// Geometric and Coordinate Transformations
NodeFactory.AddNodeAsPrototype('Vision/Geometric and Coordinate Transformations/Calibration/F_VN_CalibrateCamera', node_F_VN_CalibrateCamera);
//NodeFactory.AddNodeAsPrototype('Vision/Geometric and Coordinate Transformations/Calibration/F_VN_CalibrateCameraExp', node_F_VN_CalibrateCameraExp);
//NodeFactory.AddNodeAsPrototype('Vision/Geometric and Coordinate Transformations/Calibration/F_VN_CalibrateCameraExp2', node_F_VN_CalibrateCameraExp2);
//NodeFactory.AddNodeAsPrototype('Vision/Geometric and Coordinate Transformations/Calibration/F_VN_CalibrateCameraExp3', node_F_VN_CalibrateCameraExp3);
NodeFactory.AddNodeAsPrototype('Vision/Geometric and Coordinate Transformations/Calibration/F_VN_CalibrateCameraManually', node_F_VN_CalibrateCameraManually);
NodeFactory.AddNodeAsPrototype('Vision/Geometric and Coordinate Transformations/Calibration/F_VN_CalibrateCameraManuallyExp', node_F_VN_CalibrateCameraManuallyExp);
NodeFactory.AddNodeAsPrototype('Vision/Geometric and Coordinate Transformations/Calibration/F_VN_CalibrateCameraPlanar', node_F_VN_CalibrateCameraPlanar);
NodeFactory.AddNodeAsPrototype('Vision/Geometric and Coordinate Transformations/Calibration/F_VN_CalibrateCameraPlanarExp', node_F_VN_CalibrateCameraPlanarExp);
//NodeFactory.AddNodeAsPrototype('Vision/Geometric and Coordinate Transformations/Calibration/F_VN_CalibrateLinescanCamera', node_F_VN_CalibrateLinescanCamera);
//NodeFactory.AddNodeAsPrototype('Vision/Geometric and Coordinate Transformations/Calibration/F_VN_CalibrateLinescanCameraExp', node_F_VN_CalibrateLinescanCameraExp);
NodeFactory.AddNodeAsPrototype('Vision/Geometric and Coordinate Transformations/Calibration/F_VN_CompensateLensDistortion', node_F_VN_CompensateLensDistortion);
NodeFactory.AddNodeAsPrototype('Vision/Geometric and Coordinate Transformations/Calibration/F_VN_CompensateLensDistortionExp1', node_F_VN_CompensateLensDistortionExp1);
NodeFactory.AddNodeAsPrototype('Vision/Geometric and Coordinate Transformations/Calibration/F_VN_CompensateLensDistortionExp2', node_F_VN_CompensateLensDistortionExp2);
NodeFactory.AddNodeAsPrototype('Vision/Geometric and Coordinate Transformations/Calibration/F_VN_CompensateLensDistortionForPoints', node_F_VN_CompensateLensDistortionForPoints);
NodeFactory.AddNodeAsPrototype('Vision/Geometric and Coordinate Transformations/Calibration/F_VN_CompensateLensDistortionForPointsExp1', node_F_VN_CompensateLensDistortionForPointsExp1);
NodeFactory.AddNodeAsPrototype('Vision/Geometric and Coordinate Transformations/Calibration/F_VN_CompensateLensDistortionForPointsExp2', node_F_VN_CompensateLensDistortionForPointsExp2);
NodeFactory.AddNodeAsPrototype('Vision/Geometric and Coordinate Transformations/Calibration/F_VN_DetectPatternPoints', node_F_VN_DetectPatternPoints);
NodeFactory.AddNodeAsPrototype('Vision/Geometric and Coordinate Transformations/Calibration/F_VN_DetectPatternPointsExp', node_F_VN_DetectPatternPointsExp);
NodeFactory.AddNodeAsPrototype('Vision/Geometric and Coordinate Transformations/Calibration/F_VN_DetectPatternPoints2', node_F_VN_DetectPatternPoints2);
NodeFactory.AddNodeAsPrototype('Vision/Geometric and Coordinate Transformations/Calibration/F_VN_GenerateCalibrationPatternReferencePoints', node_F_VN_GenerateCalibrationPatternReferencePoints);
NodeFactory.AddNodeAsPrototype('Vision/Geometric and Coordinate Transformations/Calibration/F_VN_ImagePointsWorldDistance', node_F_VN_ImagePointsWorldDistance);
NodeFactory.AddNodeAsPrototype('Vision/Geometric and Coordinate Transformations/Calibration/F_VN_SolvePnP', node_F_VN_SolvePnP);
NodeFactory.AddNodeAsPrototype('Vision/Geometric and Coordinate Transformations/Calibration/F_VN_SolvePnPExp', node_F_VN_SolvePnPExp);
NodeFactory.AddNodeAsPrototype('Vision/Geometric and Coordinate Transformations/Calibration/F_VN_SortAxisAlignedPatternPoints', node_F_VN_SortAxisAlignedPatternPoints);
NodeFactory.AddNodeAsPrototype('Vision/Geometric and Coordinate Transformations/Calibration/F_VN_SortDetectedPatternPoints', node_F_VN_SortDetectedPatternPoints);
NodeFactory.AddNodeAsPrototype('Vision/Geometric and Coordinate Transformations/Calibration/F_VN_TransformCoordinatesImageToWorld_Container', node_F_VN_TransformCoordinatesImageToWorld_Container);
NodeFactory.AddNodeAsPrototype('Vision/Geometric and Coordinate Transformations/Calibration/F_VN_TransformCoordinatesImageToWorld_Point', node_F_VN_TransformCoordinatesImageToWorld_Point);
NodeFactory.AddNodeAsPrototype('Vision/Geometric and Coordinate Transformations/Calibration/F_VN_TransformCoordinatesPlanar_Container', node_F_VN_TransformCoordinatesPlanar_Container);
NodeFactory.AddNodeAsPrototype('Vision/Geometric and Coordinate Transformations/Calibration/F_VN_TransformCoordinatesPlanar_Point', node_F_VN_TransformCoordinatesPlanar_Point);
NodeFactory.AddNodeAsPrototype('Vision/Geometric and Coordinate Transformations/Calibration/F_VN_TransformCoordinatesWorldToImage_Container', node_F_VN_TransformCoordinatesWorldToImage_Container);
NodeFactory.AddNodeAsPrototype('Vision/Geometric and Coordinate Transformations/Calibration/F_VN_TransformCoordinatesWorldToImage_Point', node_F_VN_TransformCoordinatesWorldToImage_Point);
NodeFactory.AddNodeAsPrototype('Vision/Geometric and Coordinate Transformations/F_VN_AlignRotatedImageRegion', node_F_VN_AlignRotatedImageRegion);
NodeFactory.AddNodeAsPrototype('Vision/Geometric and Coordinate Transformations/F_VN_AlignRotatedImageRegionExp', node_F_VN_AlignRotatedImageRegionExp);
NodeFactory.AddNodeAsPrototype('Vision/Geometric and Coordinate Transformations/F_VN_ApplyRotationToAffineTransformation', node_F_VN_ApplyRotationToAffineTransformation);
NodeFactory.AddNodeAsPrototype('Vision/Geometric and Coordinate Transformations/F_VN_ApplyRotationToAffineTransformationExp', node_F_VN_ApplyRotationToAffineTransformationExp);
NodeFactory.AddNodeAsPrototype('Vision/Geometric and Coordinate Transformations/F_VN_ApplyScalingToAffineTransformation', node_F_VN_ApplyScalingToAffineTransformation);
NodeFactory.AddNodeAsPrototype('Vision/Geometric and Coordinate Transformations/F_VN_ApplyScalingToAffineTransformationExp', node_F_VN_ApplyScalingToAffineTransformationExp);
NodeFactory.AddNodeAsPrototype('Vision/Geometric and Coordinate Transformations/F_VN_ApplyTranslationToAffineTransformation', node_F_VN_ApplyTranslationToAffineTransformation);
NodeFactory.AddNodeAsPrototype('Vision/Geometric and Coordinate Transformations/F_VN_ApplyTranslationToAffineTransformationExp', node_F_VN_ApplyTranslationToAffineTransformationExp);
NodeFactory.AddNodeAsPrototype('Vision/Geometric and Coordinate Transformations/F_VN_ApplyYAxisInversionToAffineTransformation', node_F_VN_ApplyYAxisInversionToAffineTransformation);
NodeFactory.AddNodeAsPrototype('Vision/Geometric and Coordinate Transformations/F_VN_ApplyYAxisInversionToAffineTransformationExp', node_F_VN_ApplyYAxisInversionToAffineTransformationExp);
NodeFactory.AddNodeAsPrototype('Vision/Polarization/F_VN_DemosaicPolarizedImage', node_F_VN_DemosaicPolarizedImage);
NodeFactory.AddNodeAsPrototype('Vision/Polarization/F_VN_AngleAndDegreeOfLinearPolarization', node_F_VN_AngleAndDegreeOfLinearPolarization);
NodeFactory.AddNodeAsPrototype('Vision/Polarization/F_VN_PolarizedImageGlareReduction', node_F_VN_PolarizedImageGlareReduction);
NodeFactory.AddNodeAsPrototype('Vision/Geometric and Coordinate Transformations/F_VN_ConvertCartesianToPolarAngleImage', node_F_VN_ConvertCartesianToPolarAngleImage);
NodeFactory.AddNodeAsPrototype('Vision/Geometric and Coordinate Transformations/F_VN_ConvertCartesianToPolarAngleImageExp', node_F_VN_ConvertCartesianToPolarAngleImageExp);
NodeFactory.AddNodeAsPrototype('Vision/Geometric and Coordinate Transformations/F_VN_ConvertCartesianToPolarAngles', node_F_VN_ConvertCartesianToPolarAngles);
NodeFactory.AddNodeAsPrototype('Vision/Geometric and Coordinate Transformations/F_VN_ConvertCartesianToPolarAnglesExp', node_F_VN_ConvertCartesianToPolarAnglesExp);
NodeFactory.AddNodeAsPrototype('Vision/Geometric and Coordinate Transformations/F_VN_ConvertCartesianToPolarImages', node_F_VN_ConvertCartesianToPolarImages);
NodeFactory.AddNodeAsPrototype('Vision/Geometric and Coordinate Transformations/F_VN_ConvertCartesianToPolarImagesExp', node_F_VN_ConvertCartesianToPolarImagesExp);
NodeFactory.AddNodeAsPrototype('Vision/Geometric and Coordinate Transformations/F_VN_ConvertCartesianToPolarMagnitudeImage', node_F_VN_ConvertCartesianToPolarMagnitudeImage);
NodeFactory.AddNodeAsPrototype('Vision/Geometric and Coordinate Transformations/F_VN_ConvertCartesianToPolarMagnitudes', node_F_VN_ConvertCartesianToPolarMagnitudes);
NodeFactory.AddNodeAsPrototype('Vision/Geometric and Coordinate Transformations/F_VN_ConvertCartesianToPolarPoints', node_F_VN_ConvertCartesianToPolarPoints);
NodeFactory.AddNodeAsPrototype('Vision/Geometric and Coordinate Transformations/F_VN_ConvertCartesianToPolarPointsExp', node_F_VN_ConvertCartesianToPolarPointsExp);
NodeFactory.AddNodeAsPrototype('Vision/Geometric and Coordinate Transformations/F_VN_ConvertPolarToCartesianImages', node_F_VN_ConvertPolarToCartesianImages);
NodeFactory.AddNodeAsPrototype('Vision/Geometric and Coordinate Transformations/F_VN_ConvertPolarToCartesianImagesExp', node_F_VN_ConvertPolarToCartesianImagesExp);
NodeFactory.AddNodeAsPrototype('Vision/Geometric and Coordinate Transformations/F_VN_ConvertPolarToCartesianPoints', node_F_VN_ConvertPolarToCartesianPoints);
NodeFactory.AddNodeAsPrototype('Vision/Geometric and Coordinate Transformations/F_VN_ConvertPolarToCartesianPointsExp', node_F_VN_ConvertPolarToCartesianPointsExp);
NodeFactory.AddNodeAsPrototype('Vision/Geometric and Coordinate Transformations/F_VN_DecomposeAffineTransformation', node_F_VN_DecomposeAffineTransformation);
NodeFactory.AddNodeAsPrototype('Vision/Geometric and Coordinate Transformations/F_VN_DecomposeAffineTransformationExp', node_F_VN_DecomposeAffineTransformationExp);
NodeFactory.AddNodeAsPrototype('Vision/Geometric and Coordinate Transformations/F_VN_DecomposeHomography', node_F_VN_DecomposeHomography);
NodeFactory.AddNodeAsPrototype('Vision/Geometric and Coordinate Transformations/F_VN_DecomposeHomographyExp', node_F_VN_DecomposeHomographyExp);
NodeFactory.AddNodeAsPrototype('Vision/Geometric and Coordinate Transformations/F_VN_FlipImage', node_F_VN_FlipImage);
NodeFactory.AddNodeAsPrototype('Vision/Geometric and Coordinate Transformations/F_VN_GenerateAffineTransformationUnitMatrix2D', node_F_VN_GenerateAffineTransformationUnitMatrix2D);
NodeFactory.AddNodeAsPrototype('Vision/Geometric and Coordinate Transformations/F_VN_GetAffineTransformation', node_F_VN_GetAffineTransformation);
NodeFactory.AddNodeAsPrototype('Vision/Geometric and Coordinate Transformations/F_VN_GetAffineTransformation2D', node_F_VN_GetAffineTransformation2D);
//NodeFactory.AddNodeAsPrototype('Vision/Geometric and Coordinate Transformations/F_VN_GetAffineTransformation2DExp', node_F_VN_GetAffineTransformation2DExp);
NodeFactory.AddNodeAsPrototype('Vision/Geometric and Coordinate Transformations/F_VN_GetPerspectiveTransformation', node_F_VN_GetPerspectiveTransformation);
NodeFactory.AddNodeAsPrototype('Vision/Geometric and Coordinate Transformations/F_VN_Homography', node_F_VN_Homography);
NodeFactory.AddNodeAsPrototype('Vision/Geometric and Coordinate Transformations/F_VN_HomographyExp', node_F_VN_HomographyExp);
NodeFactory.AddNodeAsPrototype('Vision/Geometric and Coordinate Transformations/F_VN_InvertAffineTransformation', node_F_VN_InvertAffineTransformation);
NodeFactory.AddNodeAsPrototype('Vision/Geometric and Coordinate Transformations/F_VN_PerspectiveTransformation', node_F_VN_PerspectiveTransformation);
NodeFactory.AddNodeAsPrototype('Vision/Geometric and Coordinate Transformations/F_VN_PyramidDown', node_F_VN_PyramidDown);
NodeFactory.AddNodeAsPrototype('Vision/Geometric and Coordinate Transformations/F_VN_PyramidUp', node_F_VN_PyramidUp);
NodeFactory.AddNodeAsPrototype('Vision/Geometric and Coordinate Transformations/F_VN_ConvertMaps', node_F_VN_ConvertMaps);
NodeFactory.AddNodeAsPrototype('Vision/Geometric and Coordinate Transformations/F_VN_RemapImage', node_F_VN_RemapImage);
NodeFactory.AddNodeAsPrototype('Vision/Geometric and Coordinate Transformations/F_VN_RemapImageExp', node_F_VN_RemapImageExp);
NodeFactory.AddNodeAsPrototype('Vision/Geometric and Coordinate Transformations/F_VN_RemapImageToLogPolarSpace', node_F_VN_RemapImageToLogPolarSpace);
NodeFactory.AddNodeAsPrototype('Vision/Geometric and Coordinate Transformations/F_VN_RemapImageToLogPolarSpaceExp', node_F_VN_RemapImageToLogPolarSpaceExp);
NodeFactory.AddNodeAsPrototype('Vision/Geometric and Coordinate Transformations/F_VN_RemapImageToLogPolarSpaceExp2', node_F_VN_RemapImageToLogPolarSpaceExp2);
NodeFactory.AddNodeAsPrototype('Vision/Geometric and Coordinate Transformations/F_VN_RemapImageToPolarSpace', node_F_VN_RemapImageToPolarSpace);
NodeFactory.AddNodeAsPrototype('Vision/Geometric and Coordinate Transformations/F_VN_RemapImageToPolarSpaceExp', node_F_VN_RemapImageToPolarSpaceExp);
NodeFactory.AddNodeAsPrototype('Vision/Geometric and Coordinate Transformations/F_VN_RemapImageToPolarSpaceExp2', node_F_VN_RemapImageToPolarSpaceExp2);
NodeFactory.AddNodeAsPrototype('Vision/Geometric and Coordinate Transformations/F_VN_ResizeImage', node_F_VN_ResizeImage);
NodeFactory.AddNodeAsPrototype('Vision/Geometric and Coordinate Transformations/F_VN_ResizeImageExp', node_F_VN_ResizeImageExp);
NodeFactory.AddNodeAsPrototype('Vision/Geometric and Coordinate Transformations/F_VN_ResizeRegion_TcVnRectangle_DINT', node_F_VN_ResizeRegion_TcVnRectangle_DINT);
NodeFactory.AddNodeAsPrototype('Vision/Geometric and Coordinate Transformations/F_VN_RotateImage', node_F_VN_RotateImage);
NodeFactory.AddNodeAsPrototype('Vision/Geometric and Coordinate Transformations/F_VN_RotateImageExp', node_F_VN_RotateImageExp);
NodeFactory.AddNodeAsPrototype('Vision/Geometric and Coordinate Transformations/F_VN_RotateImageExp2', node_F_VN_RotateImageExp2);
NodeFactory.AddNodeAsPrototype('Vision/Geometric and Coordinate Transformations/F_VN_WarpAffine', node_F_VN_WarpAffine);
NodeFactory.AddNodeAsPrototype('Vision/Geometric and Coordinate Transformations/F_VN_WarpAffine_Container', node_F_VN_WarpAffine_Container);
NodeFactory.AddNodeAsPrototype('Vision/Geometric and Coordinate Transformations/F_VN_WarpAffine_Point', node_F_VN_WarpAffine_Point);
NodeFactory.AddNodeAsPrototype('Vision/Geometric and Coordinate Transformations/F_VN_WarpAffine_Rectangle', node_F_VN_WarpAffine_Rectangle);
NodeFactory.AddNodeAsPrototype('Vision/Geometric and Coordinate Transformations/F_VN_WarpAffineExp', node_F_VN_WarpAffineExp);
NodeFactory.AddNodeAsPrototype('Vision/Geometric and Coordinate Transformations/F_VN_WarpPerspective', node_F_VN_WarpPerspective);
NodeFactory.AddNodeAsPrototype('Vision/Geometric and Coordinate Transformations/F_VN_WarpPerspective_Container', node_F_VN_WarpPerspective_Container);
NodeFactory.AddNodeAsPrototype('Vision/Geometric and Coordinate Transformations/F_VN_WarpPerspective_Point', node_F_VN_WarpPerspective_Point);
NodeFactory.AddNodeAsPrototype('Vision/Geometric and Coordinate Transformations/F_VN_WarpPerspective_Rectangle', node_F_VN_WarpPerspective_Rectangle);
NodeFactory.AddNodeAsPrototype('Vision/Geometric and Coordinate Transformations/F_VN_WarpPerspectiveExp', node_F_VN_WarpPerspectiveExp);

// Helpers
NodeFactory.AddNodeAsPrototype('Vision/Helpers/Mux10Way_ITcVnImage', node_Mux10Way_ITcVnImage);

// Image Analysis
//NodeFactory.AddNodeAsPrototype('Vision/Image Analysis/Object Detection/F_VN_AdjustActiveContour', node_F_VN_AdjustActiveContour);
NodeFactory.AddNodeAsPrototype('Vision/Image Analysis/Object Detection/F_VN_SalientFeatures', node_F_VN_SalientFeatures);
NodeFactory.AddNodeAsPrototype('Vision/Image Analysis/Object Detection/F_VN_FindRois', node_F_VN_FindRois);
NodeFactory.AddNodeAsPrototype('Vision/Image Analysis/Object Detection/F_VN_MergeRegions', node_F_VN_MergeRegions);
NodeFactory.AddNodeAsPrototype('Vision/Image Analysis/Object Detection/F_VN_DetectBlobs', node_F_VN_DetectBlobs);
NodeFactory.AddNodeAsPrototype('Vision/Image Analysis/Object Detection/F_VN_DetectBlobsExp', node_F_VN_DetectBlobsExp);
NodeFactory.AddNodeAsPrototype('Vision/Image Analysis/Object Detection/F_VN_FindContourHierarchyExp', node_F_VN_FindContourHierarchyExp);
NodeFactory.AddNodeAsPrototype('Vision/Image Analysis/Object Detection/F_VN_FindContours', node_F_VN_FindContours);
NodeFactory.AddNodeAsPrototype('Vision/Image Analysis/Object Detection/F_VN_FindContoursExp', node_F_VN_FindContoursExp);
NodeFactory.AddNodeAsPrototype('Vision/Image Analysis/Object Detection/F_VN_FindTemplateWalsh', node_F_VN_FindTemplateWalsh);
NodeFactory.AddNodeAsPrototype('Vision/Image Analysis/Object Detection/F_VN_FindTemplateWalsh_AngleRange', node_F_VN_FindTemplateWalsh_AngleRange);
NodeFactory.AddNodeAsPrototype('Vision/Image Analysis/Object Detection/F_VN_FindTemplateWalshExp', node_F_VN_FindTemplateWalshExp);
NodeFactory.AddNodeAsPrototype('Vision/Image Analysis/Object Detection/F_VN_FindTemplateWalshExp_AngleRange', node_F_VN_FindTemplateWalshExp_AngleRange);
NodeFactory.AddNodeAsPrototype('Vision/Image Analysis/Object Detection/F_VN_HoughCircles', node_F_VN_HoughCircles);
NodeFactory.AddNodeAsPrototype('Vision/Image Analysis/Object Detection/F_VN_HoughCirclesExp', node_F_VN_HoughCirclesExp);
NodeFactory.AddNodeAsPrototype('Vision/Image Analysis/Object Detection/F_VN_HoughLines', node_F_VN_HoughLines);
//NodeFactory.AddNodeAsPrototype('Vision/Image Analysis/Object Detection/F_VN_HoughLinesExp', node_F_VN_HoughLinesExp);
NodeFactory.AddNodeAsPrototype('Vision/Image Analysis/Object Detection/F_VN_HoughLinesP', node_F_VN_HoughLinesP);
NodeFactory.AddNodeAsPrototype('Vision/Image Analysis/Object Detection/F_VN_HoughLinesPExp', node_F_VN_HoughLinesPExp);
NodeFactory.AddNodeAsPrototype('Vision/Image Analysis/Object Detection/F_VN_MatchImageHuMoments', node_F_VN_MatchImageHuMoments);
NodeFactory.AddNodeAsPrototype('Vision/Image Analysis/Object Detection/F_VN_MatchTemplate', node_F_VN_MatchTemplate);
NodeFactory.AddNodeAsPrototype('Vision/Image Analysis/Object Detection/F_VN_MatchTemplateAndEvaluate', node_F_VN_MatchTemplateAndEvaluate);
NodeFactory.AddNodeAsPrototype('Vision/Image Analysis/Object Detection/F_VN_MatchTemplateWalsh', node_F_VN_MatchTemplateWalsh);
NodeFactory.AddNodeAsPrototype('Vision/Image Analysis/Object Detection/F_VN_MatchTemplateWalshExp', node_F_VN_MatchTemplateWalshExp);
NodeFactory.AddNodeAsPrototype('Vision/Image Analysis/Object Detection/F_VN_MatchTemplateAndEvaluateExp', node_F_VN_MatchTemplateAndEvaluateExp);
NodeFactory.AddNodeAsPrototype('Vision/Image Analysis/Object Detection/F_VN_MatchTemplateExp', node_F_VN_MatchTemplateExp);
NodeFactory.AddNodeAsPrototype('Vision/Image Analysis/F_VN_CannyEdgeDetection', node_F_VN_CannyEdgeDetection);
NodeFactory.AddNodeAsPrototype('Vision/Image Analysis/F_VN_CannyEdgeDetectionExp', node_F_VN_CannyEdgeDetectionExp);
NodeFactory.AddNodeAsPrototype('Vision/Image Analysis/F_VN_ConnectedComponents', node_F_VN_ConnectedComponents);
NodeFactory.AddNodeAsPrototype('Vision/Image Analysis/F_VN_ConnectedComponentsExp', node_F_VN_ConnectedComponentsExp);
NodeFactory.AddNodeAsPrototype('Vision/Image Analysis/F_VN_ConnectedComponentsWithStats', node_F_VN_ConnectedComponentsWithStats);
NodeFactory.AddNodeAsPrototype('Vision/Image Analysis/F_VN_ConnectedComponentsWithStatsExp', node_F_VN_ConnectedComponentsWithStatsExp);
NodeFactory.AddNodeAsPrototype('Vision/Image Analysis/F_VN_CountNonZeroPixels', node_F_VN_CountNonZeroPixels);
NodeFactory.AddNodeAsPrototype('Vision/Image Analysis/F_VN_DistanceTransformation', node_F_VN_DistanceTransformation);
NodeFactory.AddNodeAsPrototype('Vision/Image Analysis/F_VN_DistanceTransformationExp', node_F_VN_DistanceTransformationExp);
NodeFactory.AddNodeAsPrototype('Vision/Image Analysis/F_VN_GetConnectedComponent', node_F_VN_GetConnectedComponent);
NodeFactory.AddNodeAsPrototype('Vision/Image Analysis/F_VN_GetConnectedComponentExp', node_F_VN_GetConnectedComponentExp);
NodeFactory.AddNodeAsPrototype('Vision/Image Analysis/F_VN_ImageAverage', node_F_VN_ImageAverage);
NodeFactory.AddNodeAsPrototype('Vision/Image Analysis/F_VN_ImageAverageExp', node_F_VN_ImageAverageExp);
NodeFactory.AddNodeAsPrototype('Vision/Image Analysis/F_VN_ImageAverageStdDev', node_F_VN_ImageAverageStdDev);
NodeFactory.AddNodeAsPrototype('Vision/Image Analysis/F_VN_ImageAverageStdDevExp', node_F_VN_ImageAverageStdDevExp);
NodeFactory.AddNodeAsPrototype('Vision/Image Analysis/F_VN_ImageCenterOfMass', node_F_VN_ImageCenterOfMass);
NodeFactory.AddNodeAsPrototype('Vision/Image Analysis/F_VN_ImageCenterOfMassExp', node_F_VN_ImageCenterOfMassExp);
NodeFactory.AddNodeAsPrototype('Vision/Image Analysis/F_VN_ImageMedian', node_F_VN_ImageMedian);
NodeFactory.AddNodeAsPrototype('Vision/Image Analysis/F_VN_ImageMedianExp', node_F_VN_ImageMedianExp);
NodeFactory.AddNodeAsPrototype('Vision/Image Analysis/F_VN_ImageMoments', node_F_VN_ImageMoments);
NodeFactory.AddNodeAsPrototype('Vision/Image Analysis/F_VN_MaxPixelValue', node_F_VN_MaxPixelValue);
NodeFactory.AddNodeAsPrototype('Vision/Image Analysis/F_VN_MaxPixelValueExp', node_F_VN_MaxPixelValueExp);
NodeFactory.AddNodeAsPrototype('Vision/Image Analysis/F_VN_MinPixelValue', node_F_VN_MinPixelValue);
NodeFactory.AddNodeAsPrototype('Vision/Image Analysis/F_VN_MinPixelValueExp', node_F_VN_MinPixelValueExp);
NodeFactory.AddNodeAsPrototype('Vision/Image Analysis/F_VN_RegionOrientation', node_F_VN_RegionOrientation);
NodeFactory.AddNodeAsPrototype('Vision/Image Analysis/F_VN_RegionOrientationExp', node_F_VN_RegionOrientationExp);
NodeFactory.AddNodeAsPrototype('Vision/Image Analysis/F_VN_ImageAbsoluteAverage', node_F_VN_ImageAbsoluteAverage);
NodeFactory.AddNodeAsPrototype('Vision/Image Analysis/F_VN_UprightInnerRectangle', node_F_VN_UprightInnerRectangle);
NodeFactory.AddNodeAsPrototype('Vision/Image Analysis/F_VN_UprightInnerRectangleExp', node_F_VN_UprightInnerRectangleExp);

// Image Color and Contrast Processing
NodeFactory.AddNodeAsPrototype('Vision/Image Color and Contrast Processing/F_VN_ApplyColorMap', node_F_VN_ApplyColorMap);
//NodeFactory.AddNodeAsPrototype('Vision/Image Color and Contrast Processing/F_VN_ApplyLut', node_F_VN_ApplyLut);
NodeFactory.AddNodeAsPrototype('Vision/Image Color and Contrast Processing/F_VN_Clahe', node_F_VN_Clahe);
NodeFactory.AddNodeAsPrototype('Vision/Image Color and Contrast Processing/F_VN_ClaheExp', node_F_VN_ClaheExp);
NodeFactory.AddNodeAsPrototype('Vision/Image Color and Contrast Processing/F_VN_ConvertColorSpace', node_F_VN_ConvertColorSpace);
NodeFactory.AddNodeAsPrototype('Vision/Image Color and Contrast Processing/F_VN_GenerateColorMap', node_F_VN_GenerateColorMap);
NodeFactory.AddNodeAsPrototype('Vision/Image Color and Contrast Processing/F_VN_GenerateCustomColorMap', node_F_VN_GenerateCustomColorMap);
NodeFactory.AddNodeAsPrototype('Vision/Image Color and Contrast Processing/F_VN_Histogram', node_F_VN_Histogram);
NodeFactory.AddNodeAsPrototype('Vision/Image Color and Contrast Processing/F_VN_HistogramEqualization', node_F_VN_HistogramEqualization);
NodeFactory.AddNodeAsPrototype('Vision/Image Color and Contrast Processing/F_VN_HistogramEqualizationExp', node_F_VN_HistogramEqualizationExp);
NodeFactory.AddNodeAsPrototype('Vision/Image Color and Contrast Processing/F_VN_HistogramExp', node_F_VN_HistogramExp);
NodeFactory.AddNodeAsPrototype('Vision/Image Color and Contrast Processing/F_VN_InvertImageColor', node_F_VN_InvertImageColor);
NodeFactory.AddNodeAsPrototype('Vision/Image Color and Contrast Processing/F_VN_InvertImageColorExp', node_F_VN_InvertImageColorExp);
NodeFactory.AddNodeAsPrototype('Vision/Image Color and Contrast Processing/F_VN_NormalizeImage', node_F_VN_NormalizeImage);
NodeFactory.AddNodeAsPrototype('Vision/Image Color and Contrast Processing/F_VN_NormalizeImageExp', node_F_VN_NormalizeImageExp);
NodeFactory.AddNodeAsPrototype('Vision/Image Color and Contrast Processing/F_VN_NormalizeImageForDisplay', node_F_VN_NormalizeImageForDisplay);
//NodeFactory.AddNodeAsPrototype('Vision/Image Color and Contrast Processing/F_VN_ReferenceColorSimilarity_ITcVnColorModel', node_F_VN_ReferenceColorSimilarity_ITcVnColorModel);
//NodeFactory.AddNodeAsPrototype('Vision/Image Color and Contrast Processing/F_VN_ReferenceColorSimilarity_ITcVnMlModel', node_F_VN_ReferenceColorSimilarity_ITcVnMlModel);
NodeFactory.AddNodeAsPrototype('Vision/Image Color and Contrast Processing/F_VN_ReferenceColorSimilarity_TcVnVector3_LREAL', node_F_VN_ReferenceColorSimilarity_TcVnVector3_LREAL);
//NodeFactory.AddNodeAsPrototype('Vision/Image Color and Contrast Processing/F_VN_ReferenceColorSimilarityExp_ITcVnColorModel', node_F_VN_ReferenceColorSimilarityExp_ITcVnColorModel);
//NodeFactory.AddNodeAsPrototype('Vision/Image Color and Contrast Processing/F_VN_ReferenceColorSimilarityExp_ITcVnMlModel', node_F_VN_ReferenceColorSimilarityExp_ITcVnMlModel);
NodeFactory.AddNodeAsPrototype('Vision/Image Color and Contrast Processing/F_VN_ReferenceColorSimilarityExp_TcVnVector3_LREAL', node_F_VN_ReferenceColorSimilarityExp_TcVnVector3_LREAL);
//NodeFactory.AddNodeAsPrototype('Vision/Image Color and Contrast Processing/F_VN_TrainImageColor', node_F_VN_TrainImageColor);
//NodeFactory.AddNodeAsPrototype('Vision/Image Color and Contrast Processing/F_VN_TrainImageColor_ITcVnMlModel', node_F_VN_TrainImageColor_ITcVnMlModel);
//NodeFactory.AddNodeAsPrototype('Vision/Image Color and Contrast Processing/F_VN_TrainImageColorExp', node_F_VN_TrainImageColorExp);
//NodeFactory.AddNodeAsPrototype('Vision/Image Color and Contrast Processing/F_VN_TrainImageColorExp_ITcVnMlModel', node_F_VN_TrainImageColorExp_ITcVnMlModel);
//NodeFactory.AddNodeAsPrototype('Vision/Image Color and Contrast Processing/F_VN_TrainImageColorExp2', node_F_VN_TrainImageColorExp2);
//NodeFactory.AddNodeAsPrototype('Vision/Image Color and Contrast Processing/F_VN_TrainImageColorExp2_ITcVnMlModel', node_F_VN_TrainImageColorExp2_ITcVnMlModel);
NodeFactory.AddNodeAsPrototype('Vision/Image Color and Contrast Processing/F_VN_WhiteBalance', node_F_VN_WhiteBalance);

// Image Filtering
NodeFactory.AddNodeAsPrototype('Vision/Image Filtering/F_VN_BilateralFilter', node_F_VN_BilateralFilter);
NodeFactory.AddNodeAsPrototype('Vision/Image Filtering/F_VN_BilateralFilterExp', node_F_VN_BilateralFilterExp);
NodeFactory.AddNodeAsPrototype('Vision/Image Filtering/F_VN_BoxFilter', node_F_VN_BoxFilter);
NodeFactory.AddNodeAsPrototype('Vision/Image Filtering/F_VN_BoxFilterExp', node_F_VN_BoxFilterExp);
NodeFactory.AddNodeAsPrototype('Vision/Image Filtering/F_VN_BrightBorderObjects', node_F_VN_BrightBorderObjects);
NodeFactory.AddNodeAsPrototype('Vision/Image Filtering/F_VN_CreateStructuringElement', node_F_VN_CreateStructuringElement);
//NodeFactory.AddNodeAsPrototype('Vision/Image Filtering/F_VN_CustomFilter', node_F_VN_CustomFilter);
//NodeFactory.AddNodeAsPrototype('Vision/Image Filtering/F_VN_CustomFilterExp', node_F_VN_CustomFilterExp);
NodeFactory.AddNodeAsPrototype('Vision/Image Filtering/F_VN_DarkBorderObjects', node_F_VN_DarkBorderObjects);
NodeFactory.AddNodeAsPrototype('Vision/Image Filtering/F_VN_FillHoles', node_F_VN_FillHoles);
NodeFactory.AddNodeAsPrototype('Vision/Image Filtering/F_VN_GaussianFilter', node_F_VN_GaussianFilter);
NodeFactory.AddNodeAsPrototype('Vision/Image Filtering/F_VN_GaussianFilterExp', node_F_VN_GaussianFilterExp);
NodeFactory.AddNodeAsPrototype('Vision/Image Filtering/F_VN_LaplacianFilter', node_F_VN_LaplacianFilter);
NodeFactory.AddNodeAsPrototype('Vision/Image Filtering/F_VN_LaplacianFilterExp', node_F_VN_LaplacianFilterExp);
NodeFactory.AddNodeAsPrototype('Vision/Image Filtering/F_VN_LocalMaxima', node_F_VN_LocalMaxima);
NodeFactory.AddNodeAsPrototype('Vision/Image Filtering/F_VN_LocalMinima', node_F_VN_LocalMinima);
NodeFactory.AddNodeAsPrototype('Vision/Image Filtering/F_VN_MedianFilter', node_F_VN_MedianFilter);
NodeFactory.AddNodeAsPrototype('Vision/Image Filtering/F_VN_MorphologicalOperator', node_F_VN_MorphologicalOperator);
NodeFactory.AddNodeAsPrototype('Vision/Image Filtering/F_VN_RemoveLocalMaxima', node_F_VN_RemoveLocalMaxima);
NodeFactory.AddNodeAsPrototype('Vision/Image Filtering/F_VN_RemoveLocalMinima', node_F_VN_RemoveLocalMinima);
NodeFactory.AddNodeAsPrototype('Vision/Image Filtering/F_VN_ScharrFilter', node_F_VN_ScharrFilter);
NodeFactory.AddNodeAsPrototype('Vision/Image Filtering/F_VN_ScharrFilterExp', node_F_VN_ScharrFilterExp);
//NodeFactory.AddNodeAsPrototype('Vision/Image Filtering/F_VN_SeparableCustomFilter', node_F_VN_SeparableCustomFilter);
//NodeFactory.AddNodeAsPrototype('Vision/Image Filtering/F_VN_SeparableCustomFilterExp', node_F_VN_SeparableCustomFilterExp);
NodeFactory.AddNodeAsPrototype('Vision/Image Filtering/F_VN_SobelFilter', node_F_VN_SobelFilter);
NodeFactory.AddNodeAsPrototype('Vision/Image Filtering/F_VN_SobelFilterExp', node_F_VN_SobelFilterExp);
NodeFactory.AddNodeAsPrototype('Vision/Image Filtering/F_VN_VarianceFilter', node_F_VN_VarianceFilter);
NodeFactory.AddNodeAsPrototype('Vision/Image Filtering/F_VN_VarianceFilterExp', node_F_VN_VarianceFilterExp);
    
// Image Segmentation
NodeFactory.AddNodeAsPrototype('Vision/Image Segmentation/F_VN_AdaptiveThreshold', node_F_VN_AdaptiveThreshold);
NodeFactory.AddNodeAsPrototype('Vision/Image Segmentation/F_VN_AdaptiveThresholdExp', node_F_VN_AdaptiveThresholdExp);
NodeFactory.AddNodeAsPrototype('Vision/Image Segmentation/F_VN_CheckColorRange', node_F_VN_CheckColorRange);
NodeFactory.AddNodeAsPrototype('Vision/Image Segmentation/F_VN_DoubleThreshold', node_F_VN_DoubleThreshold);
NodeFactory.AddNodeAsPrototype('Vision/Image Segmentation/F_VN_Threshold', node_F_VN_Threshold);
NodeFactory.AddNodeAsPrototype('Vision/Image Segmentation/F_VN_WatershedSegmentationExp', node_F_VN_WatershedSegmentationExp);
NodeFactory.AddNodeAsPrototype('Vision/Image Segmentation/F_VN_SauvolaThreshold', node_F_VN_SauvolaThreshold);

// Keypoint Features
NodeFactory.AddNodeAsPrototype('Vision/Keypoint Features/F_VN_FilterGoodMatches', node_F_VN_FilterGoodMatches);
NodeFactory.AddNodeAsPrototype('Vision/Keypoint Features/F_VN_FindReferenceKeyPointsInImage', node_F_VN_FindReferenceKeyPointsInImage);
NodeFactory.AddNodeAsPrototype('Vision/Keypoint Features/F_VN_FindReferenceKeyPointsInImageAKAZE', node_F_VN_FindReferenceKeyPointsInImageAKAZE);
NodeFactory.AddNodeAsPrototype('Vision/Keypoint Features/F_VN_FindReferenceKeyPointsInImageAKAZEExp', node_F_VN_FindReferenceKeyPointsInImageAKAZEExp);
NodeFactory.AddNodeAsPrototype('Vision/Keypoint Features/F_VN_FindReferenceKeyPointsInImageBRISK', node_F_VN_FindReferenceKeyPointsInImageBRISK);
NodeFactory.AddNodeAsPrototype('Vision/Keypoint Features/F_VN_FindReferenceKeyPointsInImageBRISKExp', node_F_VN_FindReferenceKeyPointsInImageBRISKExp);
NodeFactory.AddNodeAsPrototype('Vision/Keypoint Features/F_VN_FindReferenceKeyPointsInImageExp', node_F_VN_FindReferenceKeyPointsInImageExp);
NodeFactory.AddNodeAsPrototype('Vision/Keypoint Features/F_VN_FindReferenceKeyPointsInImageORB', node_F_VN_FindReferenceKeyPointsInImageORB);
NodeFactory.AddNodeAsPrototype('Vision/Keypoint Features/F_VN_FindReferenceKeyPointsInImageORBExp', node_F_VN_FindReferenceKeyPointsInImageORBExp);
NodeFactory.AddNodeAsPrototype('Vision/Keypoint Features/F_VN_GetMatchCoordinates', node_F_VN_GetMatchCoordinates);
NodeFactory.AddNodeAsPrototype('Vision/Keypoint Features/F_VN_KeyPointsAGAST', node_F_VN_KeyPointsAGAST);
NodeFactory.AddNodeAsPrototype('Vision/Keypoint Features/F_VN_KeyPointsAGASTExp', node_F_VN_KeyPointsAGASTExp);
NodeFactory.AddNodeAsPrototype('Vision/Keypoint Features/F_VN_KeyPointsAndDescriptorsAKAZE', node_F_VN_KeyPointsAndDescriptorsAKAZE);
NodeFactory.AddNodeAsPrototype('Vision/Keypoint Features/F_VN_KeyPointsAndDescriptorsAKAZEExp', node_F_VN_KeyPointsAndDescriptorsAKAZEExp);
NodeFactory.AddNodeAsPrototype('Vision/Keypoint Features/F_VN_KeyPointsAndDescriptorsBRISK', node_F_VN_KeyPointsAndDescriptorsBRISK);
NodeFactory.AddNodeAsPrototype('Vision/Keypoint Features/F_VN_KeyPointsAndDescriptorsBRISKExp', node_F_VN_KeyPointsAndDescriptorsBRISKExp);
NodeFactory.AddNodeAsPrototype('Vision/Keypoint Features/F_VN_KeyPointsAndDescriptorsKAZE', node_F_VN_KeyPointsAndDescriptorsKAZE);
NodeFactory.AddNodeAsPrototype('Vision/Keypoint Features/F_VN_KeyPointsAndDescriptorsKAZEExp', node_F_VN_KeyPointsAndDescriptorsKAZEExp);
NodeFactory.AddNodeAsPrototype('Vision/Keypoint Features/F_VN_KeyPointsAndDescriptorsORB', node_F_VN_KeyPointsAndDescriptorsORB);
NodeFactory.AddNodeAsPrototype('Vision/Keypoint Features/F_VN_KeyPointsAndDescriptorsORBExp', node_F_VN_KeyPointsAndDescriptorsORBExp);
NodeFactory.AddNodeAsPrototype('Vision/Keypoint Features/F_VN_KeyPointsFAST', node_F_VN_KeyPointsFAST);
NodeFactory.AddNodeAsPrototype('Vision/Keypoint Features/F_VN_KeyPointsFASTExp', node_F_VN_KeyPointsFASTExp);
NodeFactory.AddNodeAsPrototype('Vision/Keypoint Features/F_VN_KeyPointsGFTT', node_F_VN_KeyPointsGFTT);
NodeFactory.AddNodeAsPrototype('Vision/Keypoint Features/F_VN_KeyPointsGFTTExp', node_F_VN_KeyPointsGFTTExp);
NodeFactory.AddNodeAsPrototype('Vision/Keypoint Features/F_VN_KeyPointsMSER', node_F_VN_KeyPointsMSER);
NodeFactory.AddNodeAsPrototype('Vision/Keypoint Features/F_VN_KeyPointsMSERExp', node_F_VN_KeyPointsMSERExp);
NodeFactory.AddNodeAsPrototype('Vision/Keypoint Features/F_VN_KeyPointsSB', node_F_VN_KeyPointsSB);
NodeFactory.AddNodeAsPrototype('Vision/Keypoint Features/F_VN_KeyPointsSBExp', node_F_VN_KeyPointsSBExp);
NodeFactory.AddNodeAsPrototype('Vision/Keypoint Features/F_VN_MatchDescriptorsBF', node_F_VN_MatchDescriptorsBF);
NodeFactory.AddNodeAsPrototype('Vision/Keypoint Features/F_VN_MatchDescriptorsBFExp', node_F_VN_MatchDescriptorsBFExp);
NodeFactory.AddNodeAsPrototype('Vision/Keypoint Features/F_VN_MatchDescriptorsFlannLsh', node_F_VN_MatchDescriptorsFlannLsh);
NodeFactory.AddNodeAsPrototype('Vision/Keypoint Features/F_VN_MatchDescriptorsFlannLshExp', node_F_VN_MatchDescriptorsFlannLshExp);
NodeFactory.AddNodeAsPrototype('Vision/Keypoint Features/F_VN_MatchDescriptorsKnnBF', node_F_VN_MatchDescriptorsKnnBF);
NodeFactory.AddNodeAsPrototype('Vision/Keypoint Features/F_VN_MatchDescriptorsKnnBFExp', node_F_VN_MatchDescriptorsKnnBFExp);
NodeFactory.AddNodeAsPrototype('Vision/Keypoint Features/F_VN_MatchDescriptorsKnnFlannLsh', node_F_VN_MatchDescriptorsKnnFlannLsh);
NodeFactory.AddNodeAsPrototype('Vision/Keypoint Features/F_VN_MatchDescriptorsKnnFlannLshExp', node_F_VN_MatchDescriptorsKnnFlannLshExp);
NodeFactory.AddNodeAsPrototype('Vision/Keypoint Features/F_VN_RegionsMSER', node_F_VN_RegionsMSER);
NodeFactory.AddNodeAsPrototype('Vision/Keypoint Features/F_VN_RegionsMSERExp', node_F_VN_RegionsMSERExp);

// Machine Learning
//NodeFactory.AddNodeAsPrototype('Vision/Machine Learning/F_VN_CreateBoostClassifier', node_F_VN_CreateBoostClassifier);
//NodeFactory.AddNodeAsPrototype('Vision/Machine Learning/F_VN_CreateBoostClassifierExp', node_F_VN_CreateBoostClassifierExp);
//NodeFactory.AddNodeAsPrototype('Vision/Machine Learning/F_VN_CreateBoostClassifierExp2', node_F_VN_CreateBoostClassifierExp2);
//NodeFactory.AddNodeAsPrototype('Vision/Machine Learning/F_VN_CreateKmppModel', node_F_VN_CreateKmppModel);
//NodeFactory.AddNodeAsPrototype('Vision/Machine Learning/F_VN_CreateKmppModelExp', node_F_VN_CreateKmppModelExp);
//NodeFactory.AddNodeAsPrototype('Vision/Machine Learning/F_VN_CreateKnnModel', node_F_VN_CreateKnnModel);
//NodeFactory.AddNodeAsPrototype('Vision/Machine Learning/F_VN_CreateLbgModel', node_F_VN_CreateLbgModel);
//NodeFactory.AddNodeAsPrototype('Vision/Machine Learning/F_VN_CreateLbgModelExp', node_F_VN_CreateLbgModelExp);
//NodeFactory.AddNodeAsPrototype('Vision/Machine Learning/F_VN_CreateLdaTransform', node_F_VN_CreateLdaTransform);
//NodeFactory.AddNodeAsPrototype('Vision/Machine Learning/F_VN_CreateLdaTransformViaComponentNum', node_F_VN_CreateLdaTransformViaComponentNum);
//NodeFactory.AddNodeAsPrototype('Vision/Machine Learning/F_VN_CreateNbcModel', node_F_VN_CreateNbcModel);
//NodeFactory.AddNodeAsPrototype('Vision/Machine Learning/F_VN_CreatePcaTransform', node_F_VN_CreatePcaTransform);
//NodeFactory.AddNodeAsPrototype('Vision/Machine Learning/F_VN_CreatePcaTransformViaComponentNum', node_F_VN_CreatePcaTransformViaComponentNum);
//NodeFactory.AddNodeAsPrototype('Vision/Machine Learning/F_VN_CreatePcaTransformViaVariance', node_F_VN_CreatePcaTransformViaVariance);
//NodeFactory.AddNodeAsPrototype('Vision/Machine Learning/F_VN_CreateRTreesModel', node_F_VN_CreateRTreesModel);
//NodeFactory.AddNodeAsPrototype('Vision/Machine Learning/F_VN_CreateRTreesModelExp', node_F_VN_CreateRTreesModelExp);
//NodeFactory.AddNodeAsPrototype('Vision/Machine Learning/F_VN_CreateRTreesModelExp2', node_F_VN_CreateRTreesModelExp2);
//NodeFactory.AddNodeAsPrototype('Vision/Machine Learning/F_VN_CreateStaModel', node_F_VN_CreateStaModel);
//NodeFactory.AddNodeAsPrototype('Vision/Machine Learning/F_VN_CreateStaModelExp', node_F_VN_CreateStaModelExp);
//NodeFactory.AddNodeAsPrototype('Vision/Machine Learning/F_VN_CreateStaModelExp2', node_F_VN_CreateStaModelExp2);
//NodeFactory.AddNodeAsPrototype('Vision/Machine Learning/F_VN_CreateSvmModel', node_F_VN_CreateSvmModel);
//NodeFactory.AddNodeAsPrototype('Vision/Machine Learning/F_VN_CreateSvmModelExp', node_F_VN_CreateSvmModelExp);
//NodeFactory.AddNodeAsPrototype('Vision/Machine Learning/F_VN_CreateSvmModelExp2', node_F_VN_CreateSvmModelExp2);
//NodeFactory.AddNodeAsPrototype('Vision/Machine Learning/F_VN_CreateSvmSgdClassifier', node_F_VN_CreateSvmSgdClassifier);
//NodeFactory.AddNodeAsPrototype('Vision/Machine Learning/F_VN_CreateSvmSgdClassifierExp', node_F_VN_CreateSvmSgdClassifierExp);
//NodeFactory.AddNodeAsPrototype('Vision/Machine Learning/F_VN_FeatureScaling', node_F_VN_FeatureScaling);
//NodeFactory.AddNodeAsPrototype('Vision/Machine Learning/F_VN_FeatureScalingExp', node_F_VN_FeatureScalingExp);
//NodeFactory.AddNodeAsPrototype('Vision/Machine Learning/F_VN_FeatureTransform', node_F_VN_FeatureTransform);
//NodeFactory.AddNodeAsPrototype('Vision/Machine Learning/F_VN_GetBatchClusters', node_F_VN_GetBatchClusters);
//NodeFactory.AddNodeAsPrototype('Vision/Machine Learning/F_VN_GetBatchClustersExp', node_F_VN_GetBatchClustersExp);
//NodeFactory.AddNodeAsPrototype('Vision/Machine Learning/F_VN_GetBatchNovelties', node_F_VN_GetBatchNovelties);
//NodeFactory.AddNodeAsPrototype('Vision/Machine Learning/F_VN_GetClusterCenter', node_F_VN_GetClusterCenter);
//NodeFactory.AddNodeAsPrototype('Vision/Machine Learning/F_VN_GetClusterNum', node_F_VN_GetClusterNum);
//NodeFactory.AddNodeAsPrototype('Vision/Machine Learning/F_VN_GetFeatureScales', node_F_VN_GetFeatureScales);
//NodeFactory.AddNodeAsPrototype('Vision/Machine Learning/F_VN_GetSampleCluster', node_F_VN_GetSampleCluster);
//NodeFactory.AddNodeAsPrototype('Vision/Machine Learning/F_VN_GetSampleClusterExp', node_F_VN_GetSampleClusterExp);
//NodeFactory.AddNodeAsPrototype('Vision/Machine Learning/F_VN_GetSampleNovelty', node_F_VN_GetSampleNovelty);
//NodeFactory.AddNodeAsPrototype('Vision/Machine Learning/F_VN_InverseFeatureScaling', node_F_VN_InverseFeatureScaling);
//NodeFactory.AddNodeAsPrototype('Vision/Machine Learning/F_VN_InverseFeatureScaling_REAL', node_F_VN_InverseFeatureScaling_REAL);
//NodeFactory.AddNodeAsPrototype('Vision/Machine Learning/F_VN_InverseFeatureScalingExp', node_F_VN_InverseFeatureScalingExp);
//NodeFactory.AddNodeAsPrototype('Vision/Machine Learning/F_VN_InverseFeatureScalingExp_REAL', node_F_VN_InverseFeatureScalingExp_REAL);
//NodeFactory.AddNodeAsPrototype('Vision/Machine Learning/F_VN_InverseFeatureTransform', node_F_VN_InverseFeatureTransform);
//NodeFactory.AddNodeAsPrototype('Vision/Machine Learning/F_VN_PredictBatch', node_F_VN_PredictBatch);
//NodeFactory.AddNodeAsPrototype('Vision/Machine Learning/F_VN_PredictBatchExp', node_F_VN_PredictBatchExp);
//NodeFactory.AddNodeAsPrototype('Vision/Machine Learning/F_VN_PredictSampleClass', node_F_VN_PredictSampleClass);
//NodeFactory.AddNodeAsPrototype('Vision/Machine Learning/F_VN_PredictSampleClassExp', node_F_VN_PredictSampleClassExp);
//NodeFactory.AddNodeAsPrototype('Vision/Machine Learning/F_VN_PredictSampleScalar', node_F_VN_PredictSampleScalar);
//NodeFactory.AddNodeAsPrototype('Vision/Machine Learning/F_VN_PredictSampleScalarExp', node_F_VN_PredictSampleScalarExp);
//NodeFactory.AddNodeAsPrototype('Vision/Machine Learning/F_VN_PredictSampleVector', node_F_VN_PredictSampleVector);
//NodeFactory.AddNodeAsPrototype('Vision/Machine Learning/F_VN_PredictSampleVectorExp', node_F_VN_PredictSampleVectorExp);
//NodeFactory.AddNodeAsPrototype('Vision/Machine Learning/F_VN_TrainBatch', node_F_VN_TrainBatch);
//NodeFactory.AddNodeAsPrototype('Vision/Machine Learning/F_VN_TrainBatchClusters', node_F_VN_TrainBatchClusters);
//NodeFactory.AddNodeAsPrototype('Vision/Machine Learning/F_VN_TrainSample', node_F_VN_TrainSample);
//NodeFactory.AddNodeAsPrototype('Vision/Machine Learning/F_VN_TrainSampleClass', node_F_VN_TrainSampleClass);
//NodeFactory.AddNodeAsPrototype('Vision/Machine Learning/F_VN_TrainSampleCluster', node_F_VN_TrainSampleCluster);
//NodeFactory.AddNodeAsPrototype('Vision/Machine Learning/F_VN_TrainSampleScalar', node_F_VN_TrainSampleScalar
//NodeFactory.AddNodeAsPrototype('Vision/Machine Learning/F_VN_TrainSampleVector', node_F_VN_TrainSampleVector);

// Measurement
NodeFactory.AddNodeAsPrototype('Vision/Measurement/F_VN_AdjustSearchWindowOrientationToLinearEdge', node_F_VN_AdjustSearchWindowOrientationToLinearEdge);
NodeFactory.AddNodeAsPrototype('Vision/Measurement/F_VN_ClosestPointsBF', node_F_VN_ClosestPointsBF);
NodeFactory.AddNodeAsPrototype('Vision/Measurement/F_VN_LocateAxisAlignedEdges', node_F_VN_LocateAxisAlignedEdges);
NodeFactory.AddNodeAsPrototype('Vision/Measurement/F_VN_LocateAxisAlignedEdgesExp', node_F_VN_LocateAxisAlignedEdgesExp);
NodeFactory.AddNodeAsPrototype('Vision/Measurement/F_VN_LocateCircularArc', node_F_VN_LocateCircularArc);
NodeFactory.AddNodeAsPrototype('Vision/Measurement/F_VN_LocateCircularArcExp', node_F_VN_LocateCircularArcExp);
NodeFactory.AddNodeAsPrototype('Vision/Measurement/F_VN_LocateCircularArcExp2', node_F_VN_LocateCircularArcExp2);
NodeFactory.AddNodeAsPrototype('Vision/Measurement/F_VN_LocateEdge', node_F_VN_LocateEdge);
NodeFactory.AddNodeAsPrototype('Vision/Measurement/F_VN_LocateEdgeExp', node_F_VN_LocateEdgeExp);
NodeFactory.AddNodeAsPrototype('Vision/Measurement/F_VN_LocateEdgeExp2', node_F_VN_LocateEdgeExp2);
NodeFactory.AddNodeAsPrototype('Vision/Measurement/F_VN_LocateEdges', node_F_VN_LocateEdges);
NodeFactory.AddNodeAsPrototype('Vision/Measurement/F_VN_LocateEdgesExp', node_F_VN_LocateEdgesExp);
NodeFactory.AddNodeAsPrototype('Vision/Measurement/F_VN_LocateEdgesExp2', node_F_VN_LocateEdgesExp2);
NodeFactory.AddNodeAsPrototype('Vision/Measurement/F_VN_LocateEllipse', node_F_VN_LocateEllipse);
NodeFactory.AddNodeAsPrototype('Vision/Measurement/F_VN_LocateEllipseExp', node_F_VN_LocateEllipseExp);
NodeFactory.AddNodeAsPrototype('Vision/Measurement/F_VN_LocateEllipseExp2', node_F_VN_LocateEllipseExp2);
NodeFactory.AddNodeAsPrototype('Vision/Measurement/F_VN_MeasureAngleBetweenEdges', node_F_VN_MeasureAngleBetweenEdges);
NodeFactory.AddNodeAsPrototype('Vision/Measurement/F_VN_MeasureAngleBetweenEdgesExp', node_F_VN_MeasureAngleBetweenEdgesExp);
NodeFactory.AddNodeAsPrototype('Vision/Measurement/F_VN_MeasureAngleBetweenEdgesExp2', node_F_VN_MeasureAngleBetweenEdgesExp2);
NodeFactory.AddNodeAsPrototype('Vision/Measurement/F_VN_MeasureEdgeDistance', node_F_VN_MeasureEdgeDistance);
NodeFactory.AddNodeAsPrototype('Vision/Measurement/F_VN_MeasureEdgeDistanceExp', node_F_VN_MeasureEdgeDistanceExp);
NodeFactory.AddNodeAsPrototype('Vision/Measurement/F_VN_MeasureEdgeDistanceExp2', node_F_VN_MeasureEdgeDistanceExp2);
NodeFactory.AddNodeAsPrototype('Vision/Measurement/F_VN_MeasureMinEdgeDistance', node_F_VN_MeasureMinEdgeDistance);
NodeFactory.AddNodeAsPrototype('Vision/Measurement/F_VN_MeasureMinEdgeDistanceExp', node_F_VN_MeasureMinEdgeDistanceExp);
NodeFactory.AddNodeAsPrototype('Vision/Measurement/F_VN_MeasureMinEdgeDistanceExp2', node_F_VN_MeasureMinEdgeDistanceExp2);

// Miscellaneous
NodeFactory.AddNodeAsPrototype('Vision/Miscellaneous/F_VN_CheckFunctionInitialization', node_F_VN_CheckFunctionInitialization);
NodeFactory.AddNodeAsPrototype('Vision/Miscellaneous/F_VN_ClipLineToBoundary', node_F_VN_ClipLineToBoundary);
NodeFactory.AddNodeAsPrototype('Vision/Miscellaneous/F_VN_ClipLineToBoundary_ITcVnImage', node_F_VN_ClipLineToBoundary_ITcVnImage);
NodeFactory.AddNodeAsPrototype('Vision/Miscellaneous/F_VN_ClipLineToBoundary_TcVnRectangle_DINT', node_F_VN_ClipLineToBoundary_TcVnRectangle_DINT);
//NodeFactory.AddNodeAsPrototype('Vision/Miscellaneous/F_VN_ConvertITcUnknownToITcVnBitmapExport', node_F_VN_ConvertITcUnknownToITcVnBitmapExport);
//NodeFactory.AddNodeAsPrototype('Vision/Miscellaneous/F_VN_ConvertITcUnknownToITcVnContainer', node_F_VN_ConvertITcUnknownToITcVnContainer);
//NodeFactory.AddNodeAsPrototype('Vision/Miscellaneous/F_VN_ConvertITcUnknownToITcVnImage', node_F_VN_ConvertITcUnknownToITcVnImage);
//NodeFactory.AddNodeAsPrototype('Vision/Miscellaneous/F_VN_ConvertITcUnknownToITcVnMlModel', node_F_VN_ConvertITcUnknownToITcVnMlModel);
NodeFactory.AddNodeAsPrototype('Vision/Miscellaneous/F_VN_DeinitializeFunction', node_F_VN_DeinitializeFunction);
//NodeFactory.AddNodeAsPrototype('Vision/Miscellaneous/F_VN_GetTimestamp', node_F_VN_GetTimestamp);
NodeFactory.AddNodeAsPrototype('Vision/Miscellaneous/F_VN_HuMomentInvariants', node_F_VN_HuMomentInvariants);
//NodeFactory.AddNodeAsPrototype('Vision/Miscellaneous/F_VN_InitMatrixStruct', node_F_VN_InitMatrixStruct);
NodeFactory.AddNodeAsPrototype('Vision/Miscellaneous/F_VN_InvertMatrix3x3', node_F_VN_InvertMatrix3x3);
NodeFactory.AddNodeAsPrototype('Vision/Miscellaneous/F_VN_LineIntersectionPoint', node_F_VN_LineIntersectionPoint);
NodeFactory.AddNodeAsPrototype('Vision/Miscellaneous/F_VN_LineIntersectionPointAndAngle', node_F_VN_LineIntersectionPointAndAngle);
//NodeFactory.AddNodeAsPrototype('Vision/Miscellaneous/F_VN_MultiplyMatrices', node_F_VN_MultiplyMatrices);
NodeFactory.AddNodeAsPrototype('Vision/Miscellaneous/F_VN_OrthogonalVector_TcVnVector2_DINT', node_F_VN_OrthogonalVector_TcVnVector2_DINT);
NodeFactory.AddNodeAsPrototype('Vision/Miscellaneous/F_VN_OrthogonalVector_TcVnVector2_LREAL', node_F_VN_OrthogonalVector_TcVnVector2_LREAL);
NodeFactory.AddNodeAsPrototype('Vision/Miscellaneous/F_VN_OrthogonalVector_TcVnVector2_REAL', node_F_VN_OrthogonalVector_TcVnVector2_REAL);
NodeFactory.AddNodeAsPrototype('Vision/Miscellaneous/F_VN_PointToLineDistance_TcVnPoint2_DINT', node_F_VN_PointToLineDistance_TcVnPoint2_DINT);
NodeFactory.AddNodeAsPrototype('Vision/Miscellaneous/F_VN_PointToLineDistance_TcVnPoint2_LREAL', node_F_VN_PointToLineDistance_TcVnPoint2_LREAL);
NodeFactory.AddNodeAsPrototype('Vision/Miscellaneous/F_VN_PointToLineDistance_TcVnPoint2_REAL', node_F_VN_PointToLineDistance_TcVnPoint2_REAL);
NodeFactory.AddNodeAsPrototype('Vision/Miscellaneous/F_VN_PointToPointDirection_TcVnPoint2_DINT', node_F_VN_PointToPointDirection_TcVnPoint2_DINT);
NodeFactory.AddNodeAsPrototype('Vision/Miscellaneous/F_VN_PointToPointDirection_TcVnPoint2_LREAL', node_F_VN_PointToPointDirection_TcVnPoint2_LREAL);
NodeFactory.AddNodeAsPrototype('Vision/Miscellaneous/F_VN_PointToPointDirection_TcVnPoint2_REAL', node_F_VN_PointToPointDirection_TcVnPoint2_REAL);
NodeFactory.AddNodeAsPrototype('Vision/Miscellaneous/F_VN_PointToPointDistance_TcVnPoint2_DINT', node_F_VN_PointToPointDistance_TcVnPoint2_DINT);
NodeFactory.AddNodeAsPrototype('Vision/Miscellaneous/F_VN_PointToPointDistance_TcVnPoint2_LREAL', node_F_VN_PointToPointDistance_TcVnPoint2_LREAL);
NodeFactory.AddNodeAsPrototype('Vision/Miscellaneous/F_VN_PointToPointDistance_TcVnPoint2_REAL', node_F_VN_PointToPointDistance_TcVnPoint2_REAL);
NodeFactory.AddNodeAsPrototype('Vision/Miscellaneous/F_VN_RotatedRectangleCorners', node_F_VN_RotatedRectangleCorners);
NodeFactory.AddNodeAsPrototype('Vision/Miscellaneous/F_VN_RotatedRectangleIntersection', node_F_VN_RotatedRectangleIntersection);
//NodeFactory.AddNodeAsPrototype('Vision/Miscellaneous/F_VN_SetRngSeed', node_F_VN_SetRngSeed);
//NodeFactory.AddNodeAsPrototype('Vision/Miscellaneous/F_VN_UpdateTimestamp', node_F_VN_UpdateTimestamp);

// NodeFactory.AddNodeAsPrototype('Vision/Miscellaneous/FB_VN_InitializeFunction', node_FB_VN_InitializeFunction);

// OCR
NodeFactory.AddNodeAsPrototype('Vision/OCR/F_VN_OCR', node_F_VN_OCR);
NodeFactory.AddNodeAsPrototype('Vision/OCR/F_VN_OCRExp', node_F_VN_OCRExp);

// Texture Analysis
NodeFactory.AddNodeAsPrototype('Vision/Texture Analysis/F_VN_Granulometry', node_F_VN_Granulometry);
NodeFactory.AddNodeAsPrototype('Vision/Texture Analysis/F_VN_HaralickFeatures', node_F_VN_HaralickFeatures);

// Neural Network
//NodeFactory.AddNodeAsPrototype('Vision/Neural Network/F_VN_ConvertDataLayout', node_F_VN_ConvertDataLayout);
//NodeFactory.AddNodeAsPrototype('Vision/Neural Network/F_VN_ExecuteNeuralNetwork', node_F_VN_ExecuteNeuralNetwork);
//NodeFactory.AddNodeAsPrototype('Vision/Neural Network/F_VN_ExecuteNeuralNetwork_MultiLayerOutput', node_F_VN_ExecuteNeuralNetwork_MultiLayerOutput);
//NodeFactory.AddNodeAsPrototype('Vision/Neural Network/F_VN_ExecuteNeuralNetwork_SingleLayerOutput', node_F_VN_ExecuteNeuralNetwork_SingleLayerOutput);
//NodeFactory.AddNodeAsPrototype('Vision/Neural Network/F_VN_GetNeuralNetworkLayerNames', node_F_VN_GetNeuralNetworkLayerNames);
//NodeFactory.AddNodeAsPrototype('Vision/Neural Network/F_VN_NonMaxSuppression', node_F_VN_NonMaxSuppression);
//NodeFactory.AddNodeAsPrototype('Vision/Neural Network/F_VN_NonMaxSuppressionExp', node_F_VN_NonMaxSuppressionExp);
NodeFactory.AddNodeAsPrototype('Vision/Neural Network/F_VN_Reduce', node_F_VN_Reduce);
NodeFactory.AddNodeAsPrototype('Vision/Neural Network/F_VN_ReduceArg', node_F_VN_ReduceArg);
//NodeFactory.AddNodeAsPrototype('Vision/Neural Network/F_VN_ReshapeImage', node_F_VN_ReshapeImage);
NodeFactory.AddNodeAsPrototype('Vision/Neural Network/F_VN_Sigmoid', node_F_VN_Sigmoid);
NodeFactory.AddNodeAsPrototype('Vision/Neural Network/F_VN_SigmoidExp', node_F_VN_SigmoidExp);
NodeFactory.AddNodeAsPrototype('Vision/Neural Network/F_VN_SoftMax', node_F_VN_SoftMax);
END_METHOD

END_FUNCTION_BLOCK

(* stored: Version 1.1.0.1, ProductVersion 3.1.4026.19
   POU VisionNodePack: Id {257fc325-f932-4b89-a50a-e9a0a38418f4}, SpecialFunc None
   Method RegisterWithNodeFactory: Id {9eda346d-cc38-44e9-a636-4948bc24f687} *)
